// Mitsubishi GX Works2 project: PLC6   PLC: FX3G

// global labels: Global1
VAR_GLOBAL
  Start AT X007 : BOOL;
  StartDayOn AT M0 : BOOL;
  Cream AT D1100 : REAL;
END_VAR
VAR_GLOBAL CONSTANT
  Min_Cream : REAL := 300;
END_VAR
VAR_GLOBAL
  Chocolate AT D1200 : REAL;
END_VAR
VAR_GLOBAL CONSTANT
  Min_Chocolate : REAL := 240;
END_VAR
VAR_GLOBAL
  Biscuit AT D1300 : REAL;
  StartDayOff AT M0 : BOOL;
  CreamQuantity AT D1100 : REAL;
END_VAR
VAR_GLOBAL CONSTANT
  secCounter3 : TIME := T#3s;
END_VAR
VAR_GLOBAL
  counter3sec AT TC3 : BOOL;
END_VAR
VAR_GLOBAL CONSTANT
  timer3Sec : INT := 30;
END_VAR
VAR_GLOBAL
  zeroing AT M1 : BOOL;
  Blinking AT TS1 : BOOL;
  zeroing2 AT TS2 : BOOL;
  Blink AT TC1 : BOOL;
END_VAR
VAR_GLOBAL CONSTANT
  BlinkTime : INT := 10;
END_VAR
VAR_GLOBAL
  Blink2 AT TC2 : BOOL;
END_VAR
VAR_GLOBAL CONSTANT
  BlinkTime2 : INT := 10;
END_VAR
VAR_GLOBAL
  Fektivi AT M2 : BOOL;
  BlinkingLamb AT M3 : BOOL;
  EndDay AT X001 : BOOL;
  TS3 AT TS3 : BOOL;
  Blinking3 AT TS3 : BOOL;
  EndBlink AT M4 : BOOL;
  StartZiluf AT X011 : BOOL;
  CreamToZiluf AT D2100 : REAL;
  fromStockToZiluf AT M5 : BOOL;
END_VAR
VAR_GLOBAL CONSTANT
  Min_Biscuit : REAL := 6;
END_VAR
VAR_GLOBAL
  BiscuitToZiluf AT D2200 : REAL;
  Start_MachineA AT X010 : BOOL;
  close_MachineA AT X005 : BOOL;
  MachineA_ON AT M6 : BOOL;
  Sen_15 AT X002 : BOOL;
  Sen_30 AT X001 : BOOL;
  Ziluf_System AT M7 : BOOL;
  Ziluf_End AT M8 : BOOL;
  camreON AT X003 : BOOL;
  Ziluf_LampON AT Y004 : BOOL;
  EndBlink2 AT M23 : BOOL;
  zeroing1 AT M11 : BOOL;
  Blinking2 AT TS4 : BOOL;
  BlinkingLamp AT M21 : BOOL;
  Blink3 AT TC4 : BOOL;
END_VAR
VAR_GLOBAL CONSTANT
  BlinkTime3 : INT := 10;
END_VAR
VAR_GLOBAL
  zeroing12 AT TS5 : BOOL;
  BlinkingLamp2 AT M22 : BOOL;
  Blink4 AT TC5 : BOOL;
END_VAR
VAR_GLOBAL CONSTANT
  BlinkTime4 : INT := 10;
END_VAR
VAR_GLOBAL
  counter4sec AT TC6 : BOOL;
END_VAR
VAR_GLOBAL CONSTANT
  timer4sec : INT := 40;
END_VAR
VAR_GLOBAL
  Blinking4 AT TS6 : BOOL;
  DipChocolate AT X006 : BOOL;
  analog_input1 AT D8280 : INT;
END_VAR
VAR_GLOBAL CONSTANT
  UpperBound : REAL := 5;
  LowerBound : REAL := 1.0;
END_VAR
VAR_GLOBAL
  CheckIfLowerThan5 AT M30 : BOOL;
END_VAR
VAR_GLOBAL CONSTANT
  Normalization : REAL := 399.0;
END_VAR
VAR_GLOBAL
  NormalAnalogValue AT D8290 : REAL;
END_VAR
VAR_GLOBAL CONSTANT
  UpperBound10 : REAL := 10;
  UpperBound5 : REAL := 5;
END_VAR
VAR_GLOBAL
  CheckLowerThan10 AT M31 : BOOL;
END_VAR
VAR_GLOBAL CONSTANT
  RegularKrembo : REAL := 120.0;
END_VAR
VAR_GLOBAL
  DipChocolateContainer AT D2200 : REAL;
END_VAR
VAR_GLOBAL CONSTANT
  DoubleKrembo : REAL := 240;
  Counter5sec : INT := 50;
END_VAR
VAR_GLOBAL
  Timer5sec AT TC7 : BOOL;
  save_analog2Value AT D8400 : REAL;
  save_analog1Value AT D8350 : INT;
  DipLamp AT TS7 : BOOL;
  DipLampON AT M40 : BOOL;
  CheckIGreaterThan5 AT M31 : BOOL;
  DipLampONFor5Sec AT M50 : BOOL;
  PacKrembo AT X000 : BOOL;
END_VAR
VAR_GLOBAL CONSTANT
  FivePac : INT := 5;
END_VAR
VAR_GLOBAL
  counter5Krembos AT CC1 : BOOL;
  count5krembos AT CS1 : BOOL;
  Fektivi5KremboON AT M55 : BOOL;
  counter6Krembos AT CC2 : BOOL;
END_VAR
VAR_GLOBAL CONSTANT
  SixPac : INT := 6;
END_VAR
VAR_GLOBAL
  count6krembos AT CS2 : BOOL;
  LampForPackgingon AT M60 : BOOL;
  KrembosContainer AT D1111 : REAL;
END_VAR
VAR_GLOBAL CONSTANT
  ADD6Krembos : REAL := 6;
  ADDKrembo : REAL := 1;
  Halek10 : REAL := 10;
END_VAR
VAR_GLOBAL
  CountKrembosENDDAY AT D1115 : REAL;
END_VAR
VAR_GLOBAL CONSTANT
  MulFourty : INT := 40;
END_VAR
VAR_GLOBAL
  analogOutput AT D8282 : INT;
  LampY7 AT Y007 : BOOL;
  LampY0 AT Y000 : BOOL;
  LampY1 AT Y001 : BOOL;
  LampY3 AT Y003 : BOOL;
  LampY2 AT Y002 : BOOL;
  LampAllDay AT M70 : BOOL;
  CheckContainers AT M69 : BOOL;
  count6 AT CN2 : INT;
  CheckDone AT M68 : BOOL;
  FektiviY7 AT M80 : BOOL;
  closeMachineA AT M61 : BOOL;
END_VAR

// task Task_01 (event TRUE, interval 0, priority 31): POU_01

PROGRAM POU_01
(* structured ladder/FBD written out as ST: instructions are called as NAME(EN, inputs, outputs); _pN, _eN, _tN stand for wires *)
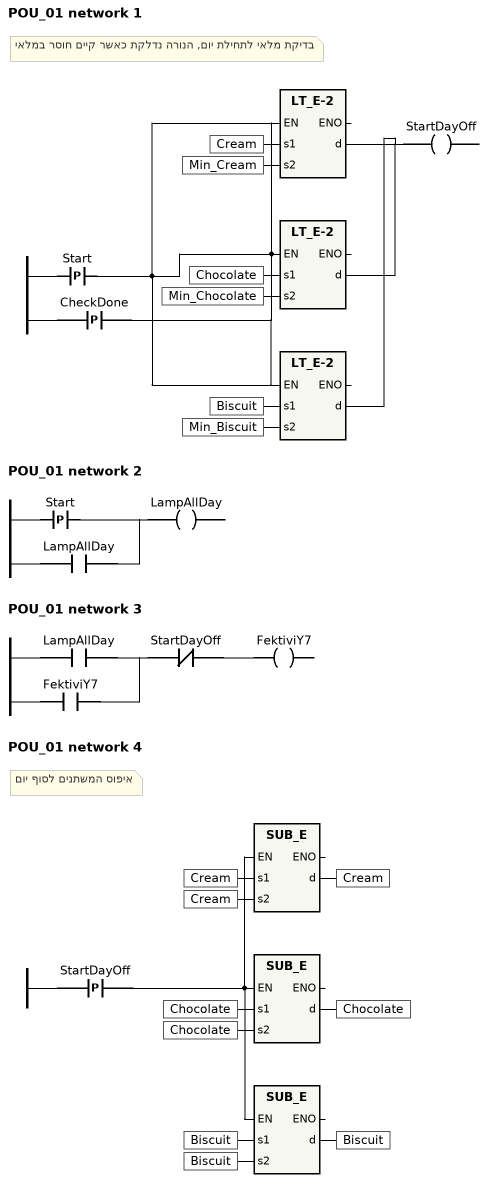
(* network 1 *)
(* בדיקת מלאי לתחילת יום, הנורה נדלקת כאשר קיים חוסר במלאי *)
_p1 := LDP(TRUE, Start) OR LDP(TRUE, CheckDone);
LT_E(_p1, Cream, Min_Cream, _t2);
LT_E(_p1, Chocolate, Min_Chocolate, _t3);
LT_E(_p1, Biscuit, Min_Biscuit, _t4);
StartDayOff := _t2 OR _t3 OR _t4;
(* network 2 *)
LampAllDay := LDP(TRUE, Start) OR LampAllDay;
(* network 3 *)
FektiviY7 := (LampAllDay OR FektiviY7) AND NOT StartDayOff;
(* network 4 *)
(* איפוס המשתנים לסוף יום *)
_p1 := LDP(TRUE, StartDayOff);
SUB_E(_p1, Cream, Cream, Cream);
SUB_E(_p1, Chocolate, Chocolate, Chocolate);
SUB_E(_p1, Biscuit, Biscuit, Biscuit);
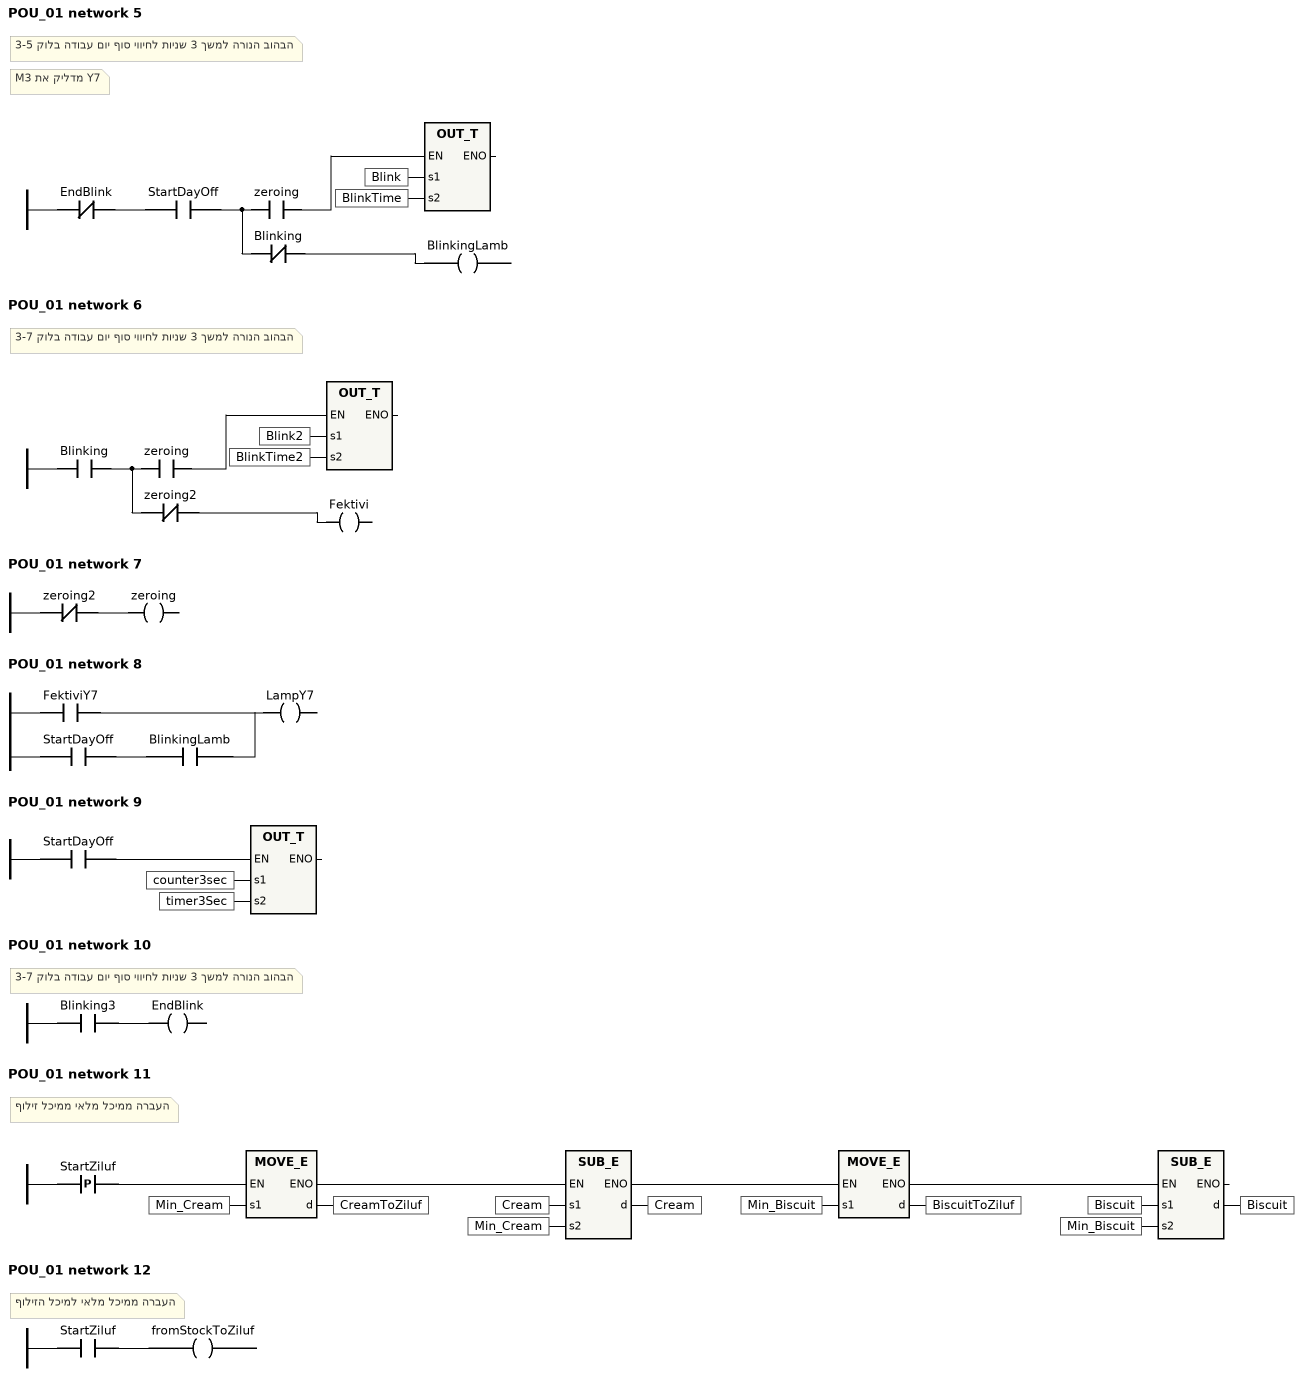
(* network 5 *)
(* הבהוב הנורה למשך 3 שניות לחיווי סוף יום עבודה בלוק 3-5 *)
(* M3 מדליק את Y7 *)
_p1 := NOT EndBlink AND StartDayOff;
OUT_T(_p1 AND zeroing, Blink, BlinkTime);
BlinkingLamb := _p1 AND NOT Blinking;
(* network 6 *)
(* הבהוב הנורה למשך 3 שניות לחיווי סוף יום עבודה בלוק 3-7 *)
OUT_T(Blinking AND zeroing, Blink2, BlinkTime2);
Fektivi := Blinking AND NOT zeroing2;
(* network 7 *)
zeroing := NOT zeroing2;
(* network 8 *)
LampY7 := FektiviY7 OR (StartDayOff AND BlinkingLamb);
(* network 9 *)
OUT_T(StartDayOff, counter3sec, timer3Sec);
(* network 10 *)
(* הבהוב הנורה למשך 3 שניות לחיווי סוף יום עבודה בלוק 3-7 *)
EndBlink := Blinking3;
(* network 11 *)
(* העברה ממיכל מלאי ממיכל זילוף *)
_e1 := MOVE_E(LDP(TRUE, StartZiluf), Min_Cream, CreamToZiluf);
_e2 := SUB_E(_e1, Cream, Min_Cream, Cream);
_e3 := MOVE_E(_e2, Min_Biscuit, BiscuitToZiluf);
SUB_E(_e3, Biscuit, Min_Biscuit, Biscuit);
(* network 12 *)
(* העברה ממיכל מלאי למיכל הזילוף *)
fromStockToZiluf := StartZiluf;
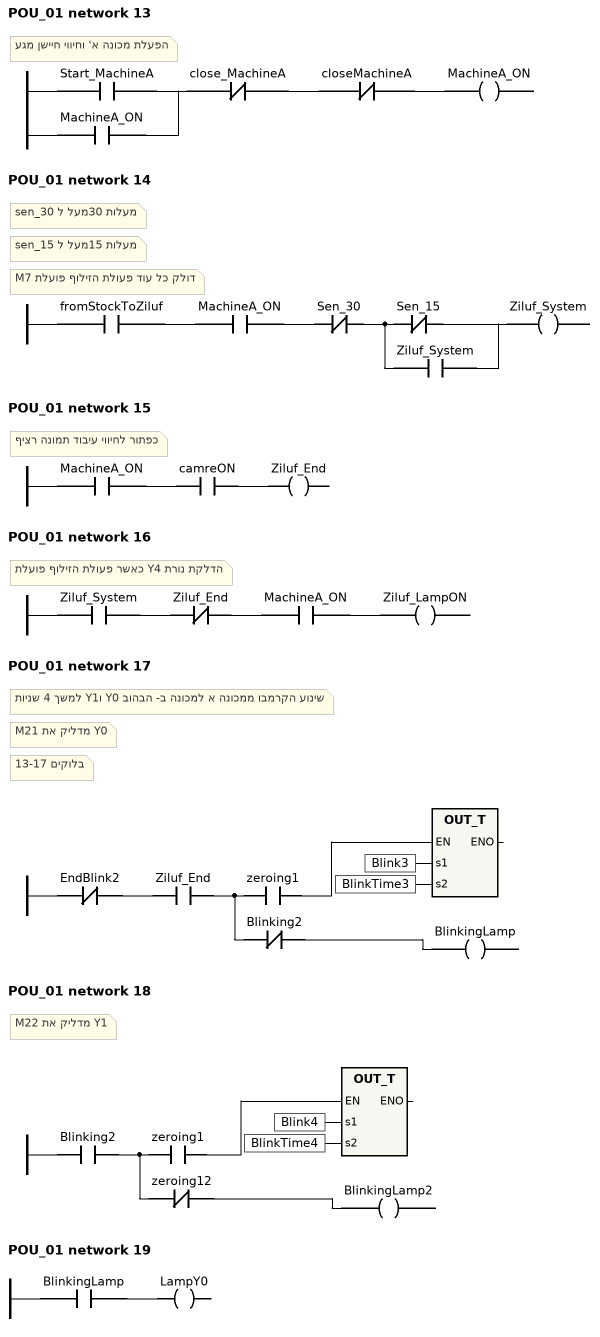
(* network 13 *)
(* הפעלת מכונה א' וחיווי חיישן מגע *)
MachineA_ON := ((Start_MachineA OR MachineA_ON) AND NOT close_MachineA) AND NOT closeMachineA;
(* network 14 *)
(* sen_30 מעל ל30 מעלות *)
(* sen_15 מעל ל15 מעלות *)
(* M7 דולק כל עוד פעולת הזילוף פועלת *)
_p1 := fromStockToZiluf AND MachineA_ON AND NOT Sen_30;
Ziluf_System := (_p1 AND NOT Sen_15) OR (_p1 AND Ziluf_System);
(* network 15 *)
(* כפתור לחיווי עיבוד תמונה רציף *)
Ziluf_End := MachineA_ON AND camreON;
(* network 16 *)
(* הדלקת נורת Y4 כאשר פעולת הזילוף פועלת *)
Ziluf_LampON := Ziluf_System AND NOT Ziluf_End AND MachineA_ON;
(* network 17 *)
(* שינוע הקרמבו ממכונה א למכונה ב- הבהוב Y0 וY1 למשך 4 שניות *)
(* M21 מדליק את Y0 *)
(* בלוקים 13-17 *)
_p1 := NOT EndBlink2 AND Ziluf_End;
OUT_T(_p1 AND zeroing1, Blink3, BlinkTime3);
BlinkingLamp := _p1 AND NOT Blinking2;
(* network 18 *)
(* M22 מדליק את Y1 *)
OUT_T(Blinking2 AND zeroing1, Blink4, BlinkTime4);
BlinkingLamp2 := Blinking2 AND NOT zeroing12;
(* network 19 *)
LampY0 := BlinkingLamp;
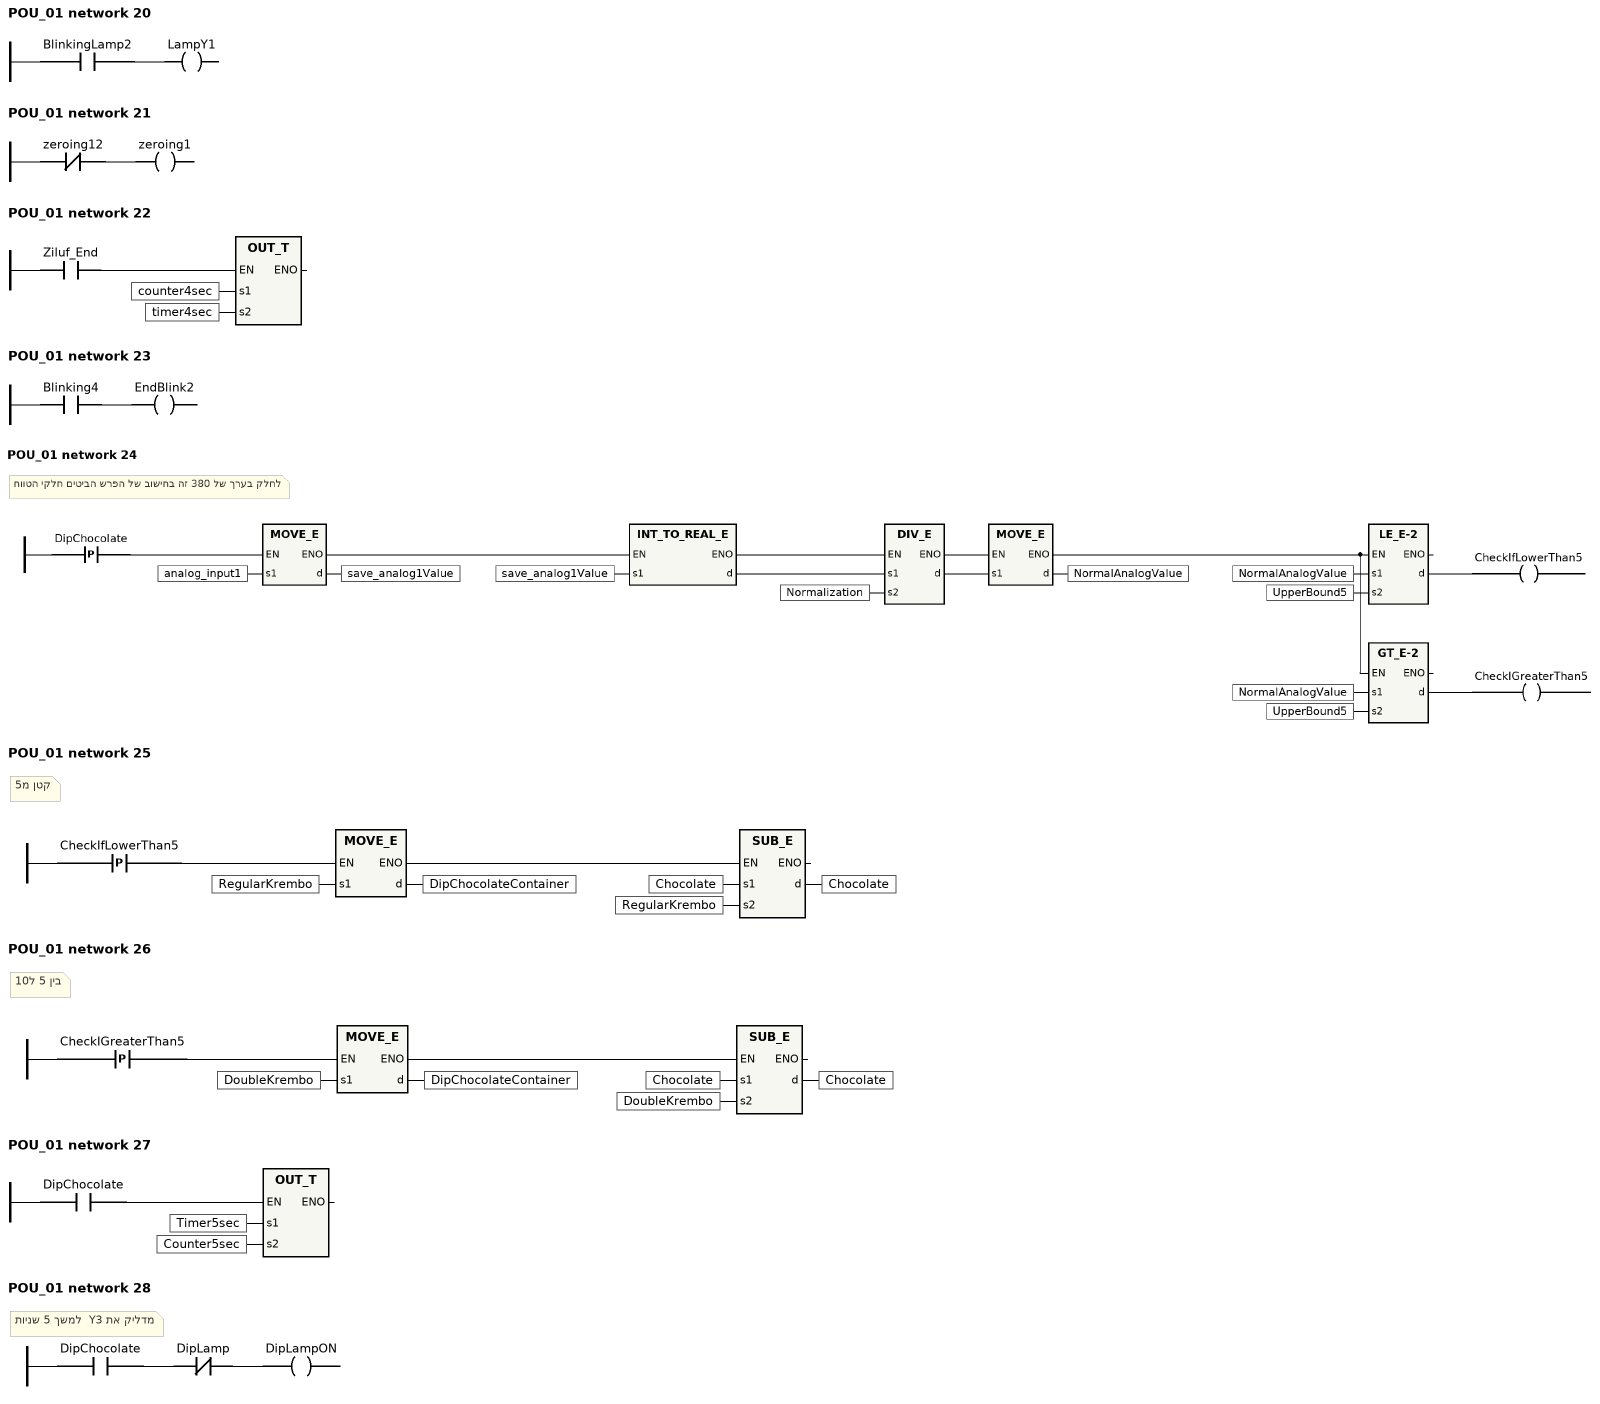
(* network 20 *)
LampY1 := BlinkingLamp2;
(* network 21 *)
zeroing1 := NOT zeroing12;
(* network 22 *)
OUT_T(Ziluf_End, counter4sec, timer4sec);
(* network 23 *)
EndBlink2 := Blinking4;
(* network 24 *)
(* לחלק בערך של 380 זה בחישוב של הפרש הביטים חלקי הטווח *)
_e1 := MOVE_E(LDP(TRUE, DipChocolate), analog_input1, save_analog1Value);
_e3 := INT_TO_REAL_E(_e1, save_analog1Value, _t2);
_e5 := DIV_E(_e3, _t2, Normalization, _t4);
_e6 := MOVE_E(_e5, _t4, NormalAnalogValue);
LE_E(_e6, NormalAnalogValue, UpperBound5, _t7);
CheckIfLowerThan5 := _t7;
GT_E(_e6, NormalAnalogValue, UpperBound5, _t8);
CheckIGreaterThan5 := _t8;
(* network 25 *)
(* קטן מ5 *)
_e1 := MOVE_E(LDP(TRUE, CheckIfLowerThan5), RegularKrembo, DipChocolateContainer);
SUB_E(_e1, Chocolate, RegularKrembo, Chocolate);
(* network 26 *)
(* בין 5 ל10 *)
_e1 := MOVE_E(LDP(TRUE, CheckIGreaterThan5), DoubleKrembo, DipChocolateContainer);
SUB_E(_e1, Chocolate, DoubleKrembo, Chocolate);
(* network 27 *)
OUT_T(DipChocolate, Timer5sec, Counter5sec);
(* network 28 *)
(* מדליק את Y3  למשך 5 שניות *)
DipLampON := DipChocolate AND NOT DipLamp;
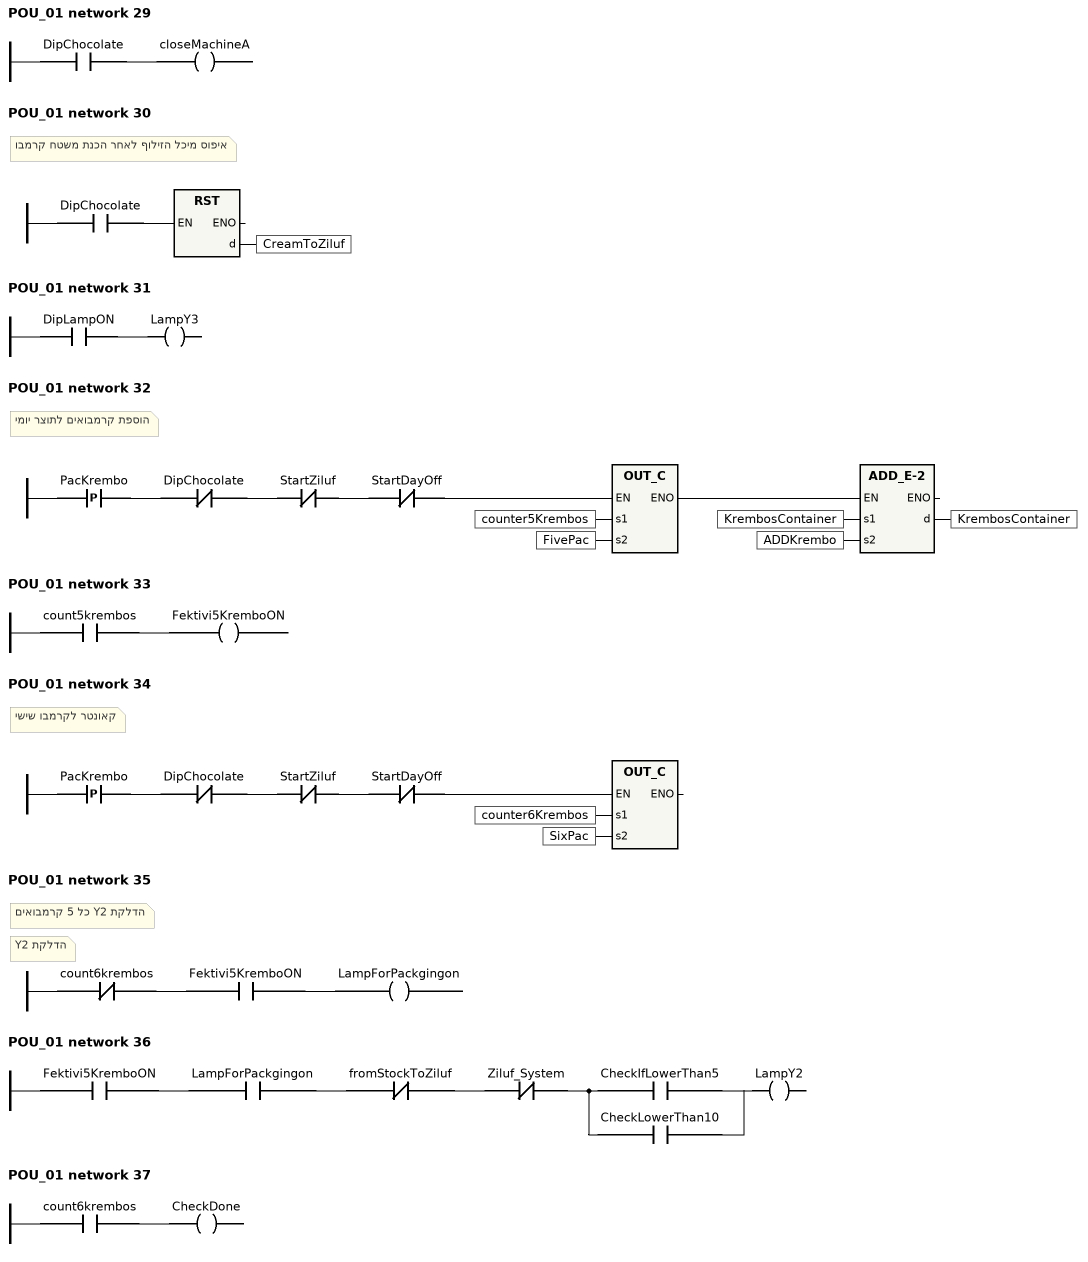
(* network 29 *)
closeMachineA := DipChocolate;
(* network 30 *)
(* איפוס מיכל הזילוף לאחר הכנת משטח קרמבו *)
RST(DipChocolate, CreamToZiluf);
(* network 31 *)
LampY3 := DipLampON;
(* network 32 *)
(* הוספת קרמבואים לתוצר יומי *)
_e1 := OUT_C(LDP(TRUE, PacKrembo) AND NOT DipChocolate AND NOT StartZiluf AND NOT StartDayOff, counter5Krembos, FivePac);
ADD_E(_e1, KrembosContainer, ADDKrembo, KrembosContainer);
(* network 33 *)
Fektivi5KremboON := count5krembos;
(* network 34 *)
(* קאונטר לקרמבו שישי *)
OUT_C(LDP(TRUE, PacKrembo) AND NOT DipChocolate AND NOT StartZiluf AND NOT StartDayOff, counter6Krembos, SixPac);
(* network 35 *)
(* הדלקת Y2 כל 5 קרמבואים *)
(* הדלקת Y2 *)
LampForPackgingon := NOT count6krembos AND Fektivi5KremboON;
(* network 36 *)
_p1 := Fektivi5KremboON AND LampForPackgingon AND NOT fromStockToZiluf AND NOT Ziluf_System;
LampY2 := (_p1 AND CheckIfLowerThan5) OR (_p1 AND CheckLowerThan10);
(* network 37 *)
CheckDone := count6krembos;
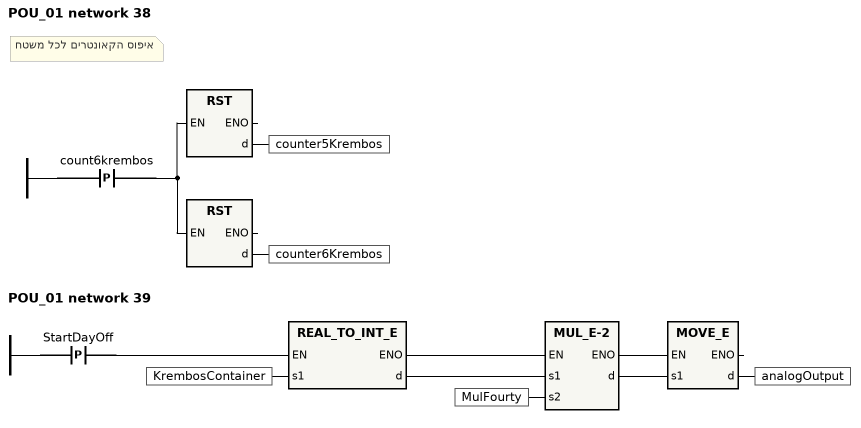
(* network 38 *)
(* איפוס הקאונטרים לכל משטח *)
_p1 := LDP(TRUE, count6krembos);
RST(_p1, counter5Krembos);
RST(_p1, counter6Krembos);
(* network 39 *)
_e2 := REAL_TO_INT_E(LDP(TRUE, StartDayOff), KrembosContainer, _t1);
_e4 := MUL_E(_e2, _t1, MulFourty, _t3);
MOVE_E(_e4, _t3, analogOutput);
END_PROGRAM
